(* IEC 61131-3 sources: programs/VI-54/VI-54_20171205/VI-54_20171205/Stations/Screen/LseClass170718/Class/ReceiveDataCMD_PLC, 1 file *)

(* ---- ReceiveDataCMD_PLC.st ---- *)
(*!
<Class
	Name               = "ReceiveDataCMD_PLC"
	Revision           = "1.0"
	RealtimeTask       = "false"
	CyclicTask         = "false"
	BackgroundTask     = "false"
	Sigmatek           = "false"
	OSInterface        = "false"
	HighPriority       = "false"
	Automatic          = "false"
	UpdateMode         = "Prescan"
	SharedCommandTable = "true"
	Objectsize         = "(676,120)"
	Comment            = "This class receives data and gives it to DiagnosticWork_PLC class.">
	<Channels>
		<Client Name="cDiagnosticWork_PLC" Required="true" Internal="false" Comment="Object channel to DiagnosticWork_PLC."/>
	</Channels>
	<RevDoku>
		<Owner Company="Sigmatek"/>
		<Dokumentation Revision="1.0" Date="2016-06-02" Author="HötAnt" Company="Sigmatek" Description="Creation"/>
	</RevDoku>
	<Network Name="ReceiveDataCMD_PLC">
		<!-- List of Components in this network -->
		<Components>
			<Object
				Name       = "_base"
				Class      = "TCPComReceive"
				Position   = "(218,120)"
				Visualized = "false">
				<Channels>
					<Server Name="ClassSvr"/>
					<Server Name="ID_Source"/>
					<Server Name="sRecvCnt"/>
					<Client Name="toDataManager"/>
				</Channels>
			</Object>
		</Components>
		<Comments>
		</Comments>
		<!-- List of Connections in this network -->
		<Connections>
			<Connection Source="this.ClassSvr" Destination="_base.ClassSvr" Vertices="(1006,210),(834,210),"/>
			<Connection Source="this.ID_Source" Destination="_base.ID_Source" Vertices="(1006,270),(834,270),"/>
			<Connection Source="this.sRecvCnt" Destination="_base.sRecvCnt" Vertices="(1006,330),(834,330),"/>
			<Connection Source="_base.toDataManager" Destination="this.toDataManager" Vertices="(218,210),(38,210),"/>
		</Connections>
		<!-- Headerfiles -->
		<Options>
		</Options>
	</Network>
</Class>
*)
#pragma using TCPComReceive

ReceiveDataCMD_PLC : CLASS
: TCPComReceive
  //Servers:
  //Clients:
	cDiagnosticWork_PLC 	: CltChCmd_DiagnosticWork_PLC;
  //Variables:
  //Functions:
				//! <Function Comment="Overwrite this method in order to receive messages including the optional CMD parameter." Name="CallBackReciverCMD"/>
	FUNCTION VIRTUAL GLOBAL CallBackReciverCMD
		VAR_INPUT
			DestinationID 	: DINT;
			SourceID 	: DINT;
			size 	: UDINT;
			pdata 	: ^USINT;
			OptCMD 	: USINT;
		END_VAR
		VAR_OUTPUT
			retcode 	: BOOL;
		END_VAR;
  //Tables:
	FUNCTION @STD
		VAR_OUTPUT
			ret_code	: CONFSTATES;
		END_VAR;
	FUNCTION GLOBAL TAB @CT_;
END_CLASS;

#pragma usingLtd DiagnosticWork_PLC

#pragma warning(disable:73);

FUNCTION VIRTUAL GLOBAL ReceiveDataCMD_PLC::CallBackReciverCMD
	VAR_INPUT
		DestinationID 	: DINT;
		SourceID 	: DINT;
		size 	: UDINT;
		pdata 	: ^USINT;
		OptCMD 	: USINT;
	END_VAR
	VAR_OUTPUT
		retcode 	: BOOL;
	END_VAR

  retcode := cDiagnosticWork_PLC.ReceivedData(size, pdata, OptCMD);

END_FUNCTION
#pragma warning(default:73);
